
// ===== library: MasterCopy "InputsMapper" =====

FUNCTION_BLOCK "InputsMapper"   // FB1, SCL
TITLE = InputsMapper
{ S7_Optimized_Access := 'TRUE' }
AUTHOR : Jesus_Alguacil
VERSION : 2.0
   VAR_INPUT
      inRawByte : Byte;
      cfgSignalData : Struct
         nSignalIndex : Array[0..7] of Int;
         bSignalNormallyOpen : Array[0..7] of Bool;
      END_STRUCT;
   END_VAR
   VAR_OUTPUT
      SignalIn0 : Bool;
      SignalIn1 : Bool;
      SignalIn2 : Bool;
      SignalIn3 : Bool;
      SignalIn4 : Bool;
      SignalIn5 : Bool;
      SignalIn6 : Bool;
      SignalIn7 : Bool;
   END_VAR
   VAR
      i : Int;
      Temp : Struct
         nSignalIndex : Array[0..7] of Int;
         inRawByte : Array[0..7] of Bool;
         bSignal : Array[0..7] of Bool;
         bSignalNormallyOpen : Array[0..7] of Bool;
      END_STRUCT;
   END_VAR
BEGIN
   (*
   // -----------------------------------------------------------------------------
   // LICENSE:
       Released under the MIT License
       Copyright (c) 2025 Jesús Alguacil
       Full license text available at:
       https://github.com/JessAlguacil/InputsMapper/blob/master/LICENSE.md
   // -----------------------------------------------------------------------------
   // Function Block: InputsMapper
   // Description   : Function responsible for mapping the physical input signals from the PLC or IO-Link modules coming
   //                 from the declared Byte TO the physical inputs AND storing them in an internal logic structure FOR use in the main program
   //                 AND signal switching, in CASE a signal is TO be switched from (NO/NC).
   // Compatibility : Siemens TIA Portal V16 or later
   // Author        : Jesús Alguacil
   // Date          : 03-06-2025
   // Version       : V2.0.1
   // -----------------------------------------------------------------------------

   // GENERAL FUNCTIONALITY:
   // - Iterates over 8 input channels using a circular index counter.
   // - Maps raw input bytes (I0.0 to I0.7) into a temporary array.
   // - Compares each input value to detect signal changes (NO/NC logic).

   // MAIN LOGIC:
   // - #i := (#i + 1) MOD 8; → circular index from 0 to 7.
   // - #Temp.nSignalIndex[#i] stores the temporary input values for current channel.
   // - #Temp.bSignalNormallyOpen[#i] configuration is applied per input channel.

   // INPUTS:
   // - (inRawByte) → Data Byte containing the logical values of the physical inputs of the (PLC or IO-Link) Example(%IB0).
   // - (cfgSignalData) → nSignalIndex → OF the hmi screen where the order OF the digital inputs can be modified.
   // -                   bSignalNormallyOpen → BOOL data containing the value from the hmi screen in which it is selected if the signal is (NO/NC).

   // OUTPUTS:
   // - (SignalIn0..SignalIn7) → Logic signals already processed into individual bits.

   // NOTES:
   // - Avoids FOR loops; uses a single index variable to reduce CPU usage.
   // - Duplicate detection requires full comparison across all channels.
   // -----------------------------------------------------------------------------
   *)

   // Counter scrolling the index
   #i := (#i + 1) MOD 8;

   // Assignment of input values to temporary variables
   #Temp.bSignalNormallyOpen[#i] := #cfgSignalData.bSignalNormallyOpen[#i];
   #Temp.nSignalIndex[#i] := #cfgSignalData.nSignalIndex[#i];

   // Assignment of the input Byte to the temporary array
   #Temp.inRawByte[0] := #inRawByte.%X0;
   #Temp.inRawByte[1] := #inRawByte.%X1;
   #Temp.inRawByte[2] := #inRawByte.%X2;
   #Temp.inRawByte[3] := #inRawByte.%X3;
   #Temp.inRawByte[4] := #inRawByte.%X4;
   #Temp.inRawByte[5] := #inRawByte.%X5;
   #Temp.inRawByte[6] := #inRawByte.%X6;
   #Temp.inRawByte[7] := #inRawByte.%X7;

   // Signal change (NO/NC) and Change of the electrical connection bit
   #Temp.bSignal[#Temp.nSignalIndex[#i]] := (#Temp.bSignalNormallyOpen[#Temp.nSignalIndex[#i]] AND #Temp.inRawByte[#i]) OR (NOT #Temp.bSignalNormallyOpen[#Temp.nSignalIndex[#i]] AND NOT #Temp.inRawByte[#i]);

   // Writing the final function values into the already filtered variables
   #SignalIn0 := #Temp.bSignal[0];
   #SignalIn1 := #Temp.bSignal[1];
   #SignalIn2 := #Temp.bSignal[2];
   #SignalIn3 := #Temp.bSignal[3];
   #SignalIn4 := #Temp.bSignal[4];
   #SignalIn5 := #Temp.bSignal[5];
   #SignalIn6 := #Temp.bSignal[6];
   #SignalIn7 := #Temp.bSignal[7];

   // END BLOCK
END_FUNCTION_BLOCK